// TIA Portal project "Using Function Keys" (V13)

(* hardware
DEVICE "S7-1200 station_1"  S7-1200 Station
   slot 0: "Rack_0"  Rack  V1.0
   slot 1: "PLC_1"  CPU 1212C AC/DC/Rly  6ES7 212-1BE40-0XB0  V4.1
DEVICE "HMI_1"  KTP400 Basic PN
   slot 0: "HMI"  HMI  6AV2 123-2DB03-0AX0  13.0.1.0
   slot 1: "HMI_RT_1"  KTP400 Basic PN  6AV2 123-2DB03-0AX0  13.0.1.0
   slot 5: "HMI_1.IE_CP_1"  PROFINET Interface
      slot 1: "PROFINET Interface_1"  PROFINET Interface
         slot 1: "Port_1"  Port
*)

// ===== PLC "PLC_1"  CPU 1212C AC/DC/Rly =====

VAR_GLOBAL   // PLC tag table "Default tag table"
   "Tag_1" AT %MD5 : DWord;
   "Tag_2" AT %MD0 : DWord;
   "Tag_4" AT %MW5 : Word;
   "Tag_3" AT %MW10 : Int;
   "Tag_5" AT %M100.0 : Bool;
   "Tag_6" AT %Q0.0 : Bool;
   "Tag_7" AT %M100.1 : Bool;
   "Tag_8" AT %Q0.1 : Bool;
   "Tag_9" AT %MD5 : Time;
   "Tag_10" AT %MD12 : Real;
   "Tag_11" AT %MW15 : Int;
   "Tag_12" AT %ID30 : DWord;
   "Tag_13" AT %MD22 : Real;
   "Tag_14" AT %MW50 : Word;
   "Tag_15" AT %Q0.2 : Bool;
   "Tag_16" AT %ID34 : DWord;
   "Tag_17" AT %MD25 : Real;
   "Tag_18" AT %MD26 : Real;
   "Fill Valve" AT %QD30 : Real;
   "Drain Valve" AT %QD34 : Real;
   "Tag_19" AT %M200.0 : Bool;
   "Tag_20" AT %M200.1 : Bool;
   "Animation bit" AT %M40.0 : Bool;
   "Clock_Byte" AT %MB300 : Byte;
   "Clock_10Hz" AT %M300.0 : Bool;
   "Clock_5Hz" AT %M300.1 : Bool;
   "Clock_2.5Hz" AT %M300.2 : Bool;
   "Clock_2Hz" AT %M300.3 : Bool;
   "Clock_1.25Hz" AT %M300.4 : Bool;
   "Clock_1Hz" AT %M300.5 : Bool;
   "Clock_0.625Hz" AT %M300.6 : Bool;
   "Clock_0.5Hz" AT %M300.7 : Bool;
   "Tag_21" AT %MB60 : Byte;
   "roller" AT %MD60 : Real;
   "roller_2" AT %MD70 : Real;
   "Tag_22" AT %MD65 : Real;
   "Tag_23" AT %MW60 : Int;
   "Tag_24" AT %MW65 : Int;
   "Down" AT %M90.0 : Bool;
   "Up" AT %M90.1 : Bool;
   "Tag_25" AT %MW75 : Int;
   "Tag_26" AT %MW78 : Int;
   "Tag_27" AT %MW80 : Int;
END_VAR

// folder: System blocks/Program resources

DATA_BLOCK "IEC_Timer_0_DB"   // DB1
{ S7_Optimized_Access := 'FALSE' }
AUTHOR : Simatic
FAMILY : IEC
NAME : IEC_TMR
VERSION : 1.0
// stored: InstanceOfName ?
"?"
BEGIN
END_DATA_BLOCK

DATA_BLOCK "IEC_Timer_0_DB_1"   // DB2
{ S7_Optimized_Access := 'FALSE' }
AUTHOR : Simatic
FAMILY : IEC
NAME : IEC_TMR
VERSION : 1.0
// stored: InstanceOfName ?
"?"
BEGIN
END_DATA_BLOCK

DATA_BLOCK "IEC_Timer_0_DB_2"   // DB3
{ S7_Optimized_Access := 'FALSE' }
AUTHOR : Simatic
FAMILY : IEC
NAME : IEC_TMR
VERSION : 1.0
// stored: InstanceOfName ?
"?"
BEGIN
END_DATA_BLOCK

DATA_BLOCK "IEC_Timer_0_DB_3"   // DB4
{ S7_Optimized_Access := 'FALSE' }
AUTHOR : Simatic
FAMILY : IEC
NAME : IEC_TMR
VERSION : 1.0
// stored: InstanceOfName ?
"?"
BEGIN
END_DATA_BLOCK

// folder: (top level)

FUNCTION "MHJ-PLC-Lab-Function-S71200" : Void   // FC1, SCL
{ S7_Optimized_Access := 'FALSE' }
VERSION : 0.1
BEGIN

   #Value := PEEK(area := 16#82,
                  dbNumber := 0,
                  byteOffset := 511);
   #Value := #Value + 1;

   POKE(area := 16#82,
        dbNumber := 0,
        byteOffset := 511,
        value := #Value);

   POKE(area := 16#81,
        dbNumber := 0,
        byteOffset := 1016,
        value := #Value_01_DW);
   POKE(area := 16#81,
        dbNumber := 0,
        byteOffset := 1020,
        value := #Value_02_DW);

   POKE(area := 16#81,
        dbNumber := 0,
        byteOffset := 511,
        value := B#16#00);

   FOR #forVal := 0 TO 120 DO
       FOR #forVal_2 := 0 TO 10 DO
           #rdTimeReturn := RD_SYS_T(#outputTime);
           #rdTimeReturn := WR_SYS_T(#outputTime);
           #rdTimeReturn := RD_SYS_T(#outputTime);
           #rdTimeReturn := WR_SYS_T(#outputTime);
       END_FOR;
       #SyncVal := PEEK(area := 16#81,
                        dbNumber := 0,
                        byteOffset := 511);
       IF #SyncVal = #CompVal THEN
           GOTO M_1;
       END_IF;
   END_FOR;
   RETURN;

   M_1:
   POKE(area := 16#81,
        dbNumber := 0,
        byteOffset := 511,
        value := B#16#0);
END_FUNCTION

ORGANIZATION_BLOCK "Main"   // OB1, LAD, ProgramCycle
TITLE = "Main Program Sweep (Cycle)"
{ S7_Optimized_Access := 'FALSE' }
VERSION : 0.1
BEGIN

REGION Network 1
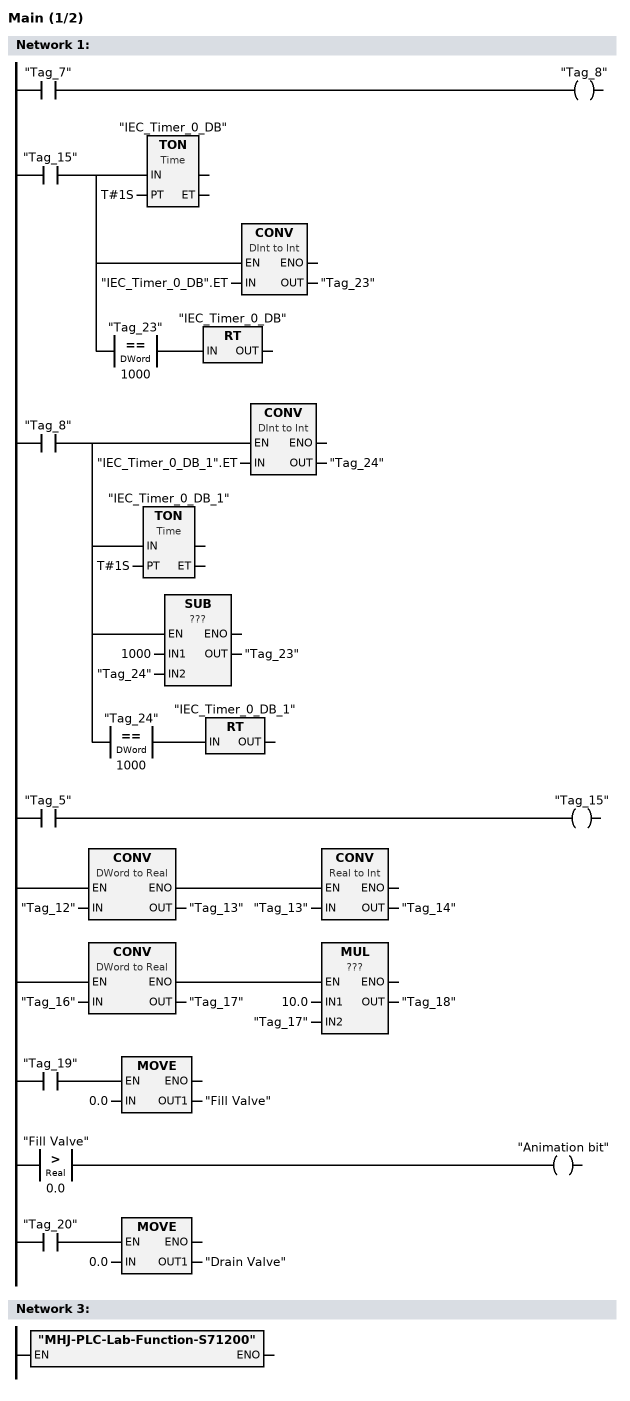
   // ENO of a box is taken as its EN; it also drops when the box reports an error
   "Tag_8" := "Tag_7";
   "IEC_Timer_0_DB".TON(IN := "Tag_15", PT := T#1S);
   IF "Tag_15" THEN "Tag_23" := DINT_TO_INT("IEC_Timer_0_DB".ET); END_IF;
   IF "Tag_15" AND ("Tag_23" = 1000) THEN RESET_TIMER("IEC_Timer_0_DB"); END_IF;
   IF "Tag_8" THEN "Tag_24" := DINT_TO_INT("IEC_Timer_0_DB_1".ET); END_IF;
   "IEC_Timer_0_DB_1".TON(IN := "Tag_8", PT := T#1S);
   IF "Tag_8" THEN "Tag_23" := 1000 - "Tag_24"; END_IF;
   IF "Tag_8" AND ("Tag_24" = 1000) THEN RESET_TIMER("IEC_Timer_0_DB_1"); END_IF;
   "Tag_15" := "Tag_5";
   "Tag_13" := DWORD_TO_REAL("Tag_12");
   "Tag_14" := REAL_TO_INT("Tag_13");
   "Tag_17" := DWORD_TO_REAL("Tag_16");
   "Tag_18" := 10.0 * "Tag_17";
   IF "Tag_19" THEN "Fill Valve" := 0.0; END_IF;
   "Animation bit" := "Fill Valve" > 0.0;
   IF "Tag_20" THEN "Drain Valve" := 0.0; END_IF;
END_REGION

REGION Network 3
   RUNG wire#powerrail
      "MHJ-PLC-Lab-Function-S71200"()
   END_RUNG
   // the same network as SCL:
   "MHJ-PLC-Lab-Function-S71200"();
END_REGION

REGION Network 4
   // Door Animation
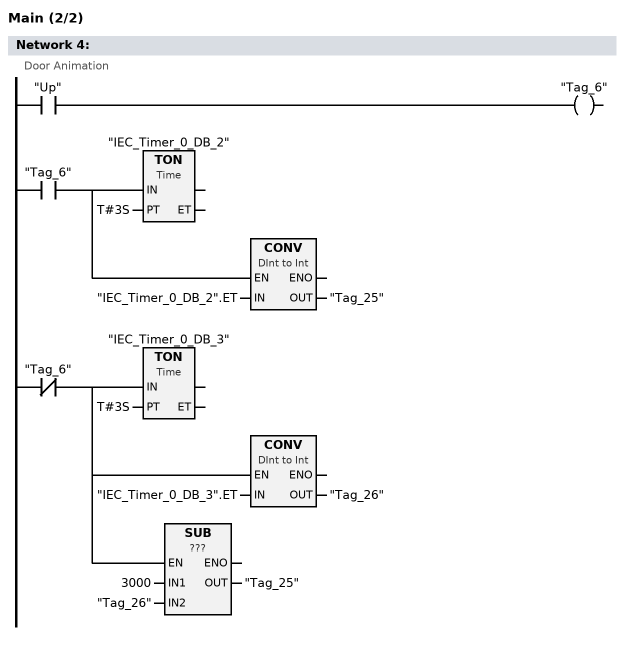
   "Tag_6" := "Up";
   "IEC_Timer_0_DB_2".TON(IN := "Tag_6", PT := T#3S);
   IF "Tag_6" THEN "Tag_25" := DINT_TO_INT("IEC_Timer_0_DB_2".ET); END_IF;
   "IEC_Timer_0_DB_3".TON(IN := NOT "Tag_6", PT := T#3S);
   IF NOT "Tag_6" THEN
       "Tag_26" := DINT_TO_INT("IEC_Timer_0_DB_3".ET);
       "Tag_25" := 3000 - "Tag_26";
   END_IF;
END_REGION
END_ORGANIZATION_BLOCK

(* ===== HMI "HMI_RT_1" =====
connection "HMI_Connection_1": ETHERNET, SMART_S7_1200_OMS

HMI tags "Default tag table"
   "Tag_5" : Bool = PLC "Tag_5", 100 ms
   "Tag_7" : Bool = PLC "Tag_7", 100 ms
   "Tag_6" : Bool = PLC "Tag_6", 100 ms
   "Tag_10" : Real = PLC "Tag_10", 1 s
   "Tag_11" : Int = PLC "Tag_11", 1 s
   "Tag_14" : Word = PLC "Tag_14", 100 ms
   "Tag_17" : Real = PLC "Tag_17", 100 ms
   "Tag_18" : Real = PLC "Tag_18", 100 ms
   "Fill Valve" : Real = PLC "Fill Valve", 100 ms
   "Drain Valve" : Real = PLC "Drain Valve", 100 ms
   "Tag_19" : Bool = PLC "Tag_19", 100 ms
   "Tag_20" : Bool = PLC "Tag_20", 100 ms
   "Animation bit" : Bool = PLC "Animation bit", 1 s
   "Tag_13" : Real = PLC "Tag_13", 1 s
   "Tag_21" : Byte = PLC "Tag_21", 100 ms
   "roller_HMI" : Real = PLC "roller", 100 ms
   "roller_2" : Real = PLC "roller_2", 100 ms
   "Tag_23" : Int = PLC "Tag_23", 100 ms
   "Tag_25" : Int = PLC "Tag_25", 100 ms
   "Up" : Bool = PLC "Up", 100 ms

graphic list "Valve": 0 'OFF'; 1..7 'Partially ON_1'; 8..10 'ON_1'

graphic list "Pipes": 0 'not flowing'; 1..7 'Partially flowing'; 8..10 'flowing'

graphic list "Roller": 0..249 '1'; 250..499 '2'; 500..749 '3'; 750..1000 '4'

graphic list "Motor": 0 'Graphic_24'; 1 'Graphic_25'

graphic list "Arrow": 0 'Graphic_27'; 1 'Graphic_26'

Template "Template_1" 480x272
   Button "Template_Button" at 388,227 size 63x44
   Button "Template_Button_3" at 28,227 size 63x44

screen "Root screen" 480x272, template "Template_1"
   Button "Button_5" at 202,139 size 122x32
   Button "Button_6" at 202,178 size 122x32
   TextField "Text field_1" at 149,97 size 224x32
   Button "Button_1" at 203,217 size 122x32
   GraphicView "Graphic view_1" at 223,8 size 83x67
   TextField "Text field_2" at 98,76 size 336x27

screen "Box" 480x272
   Button "Button_1" at 404,139 size 33x17
   Button "Button_2" at 33,139 size 33x19
   TextField "Text field_1" at 11,7 size 131x25
   Group "Group" at 33,133 size 404x46
   Button "Button_6" at 349,9 size 122x32
   Button "Button_3" at 404,236 size 67x32
   IOField "I/O field_1" at 66,109 size 39x32
   GraphicIOField "Graphic I/O field_1" at 35,170 size 32x28
   GraphicIOField "Graphic I/O field_2" at 409,170 size 32x28
   Button "Button_4" at 347,45 size 122x32

screen "Tank" 480x272
   Bar "Bar_1" at 254,70 size 120x139
   TextField "Text field_2" at 15,9 size 135x23
   GraphicView "Graphic view_1" at 254,54 size 122x18
   GraphicView "Graphic view_2" at 253,207 size 123x28
   Button "Button_4" at 429,184 size 45x23
   IOField "I/O field_1" at 383,54 size 43x29
   IOField "I/O field_2" at 383,181 size 43x29
   Button "Button_3" at 429,57 size 45x23
   IOField "I/O field_3" at 378,127 size 43x18
   GraphicView "Graphic view_5" at 295,28 size 33x28
   GraphicIOField "Graphic I/O field_1" at 387,21 size 39x32
   GraphicIOField "Graphic I/O field_2" at 385,224 size 39x32
   GraphicIOField "Graphic I/O field_3" at 327,35 size 62x13
   GraphicIOField "Graphic I/O field_4" at 424,35 size 56x13
   GraphicIOField "Graphic I/O field_5" at 325,239 size 62x13
   GraphicIOField "Graphic I/O field_6" at 422,239 size 58x13
   TextField "Text field_3" at 422,126 size 23x22
   GraphicView "Graphic view_3" at 303,233 size 23x25
   Button "Button_5" at 15,226 size 122x32
   Button "Button_1" at 15,148 size 67x32
   Button "Button_2" at 15,187 size 122x32

screen "Door" 480x272
   GraphicIOField "Graphic I/O field_1" at 10,106 size 63x27
   GraphicView "Graphic view_1" at 258,188 size 148x75
   GraphicView "Graphic view_2" at 206,106 size 44x46
   GraphicView "Graphic view_3" at 408,213 size 39x47
   Button "Button_1" at 206,158 size 41x43
   Button "Button_2" at 206,209 size 41x43
   Button "Button_3" at 406,7 size 67x32
   Button "Button_6" at 351,44 size 122x32
   Button "Button_5" at 351,84 size 122x32
   TextField "Text field_1" at 10,8 size 140x25
*)